// Mitsubishi GX Works2 project: 시퀀스 타이머 회로 1   PLC: Q03UDV

PROGRAM MAIN
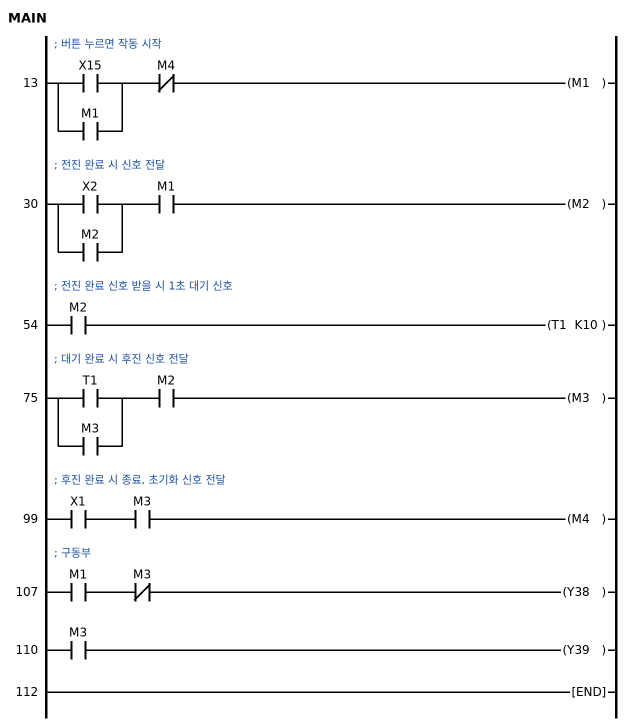
; 버튼 누르면 작동 시작
13    LD      X15
      OR      M1
      ANI     M4
      OUT     M1
; 전진 완료 시 신호 전달
30    LD      X2
      OR      M2
      AND     M1
      OUT     M2
; 전진 완료 신호 받을 시 1초 대기 신호
54    LD      M2
      OUT     T1 K10
; 대기 완료 시 후진 신호 전달
75    LD      T1
      OR      M3
      AND     M2
      OUT     M3
; 후진 완료 시 종료, 초기화 신호 전달
99    LD      X1
      AND     M3
      OUT     M4
; 구동부
107   LD      M1
      ANI     M3
      OUT     Y38
110   LD      M3
      OUT     Y39
112   END
END_PROGRAM
